Fanuc KAREL source: kt00178.KL

PROGRAM KT00178
%NOLOCKGROUP
VAR
Y1 : ARRAY[2] OF BYTE
I2:INTEGER
OUT:REAL
BEGIN
Y1[1]=2
I2=3
OUT=((Y1[1] MOD I2))
END KT00178
